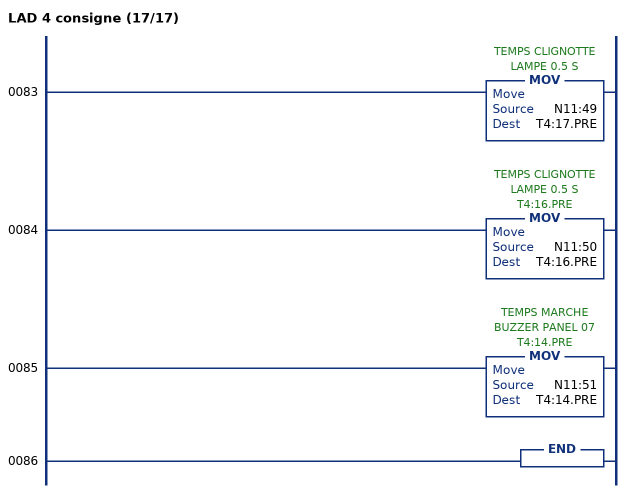
% Rung: 83 %
SOR MOV N11:49 T4:17.PRE EOR
%   N11:49  "TEMPS CLIGNOTTE LAMPE 0.5 S" %
%   T4:17.PRE  "TEMPS CLIGNOTTE LAMPE 0.5 S" %
% Rung: 84 %
SOR MOV N11:50 T4:16.PRE EOR
%   N11:50  "TEMPS CLIGNOTTE LAMPE 0.5 S" %
%   T4:16.PRE  "TEMPS CLIGNOTTE LAMPE 0.5 S T4:16.PRE" %
% Rung: 85 %
SOR MOV N11:51 T4:14.PRE EOR
%   N11:51  "TEMPS MARCHE BUZZER PANEL 07" %
%   T4:14.PRE  "TEMPS MARCHE BUZZER PANEL 07 T4:14.PRE" %
% Rung: 86 %
SOR END EOR

LADDER 5 "communicat"
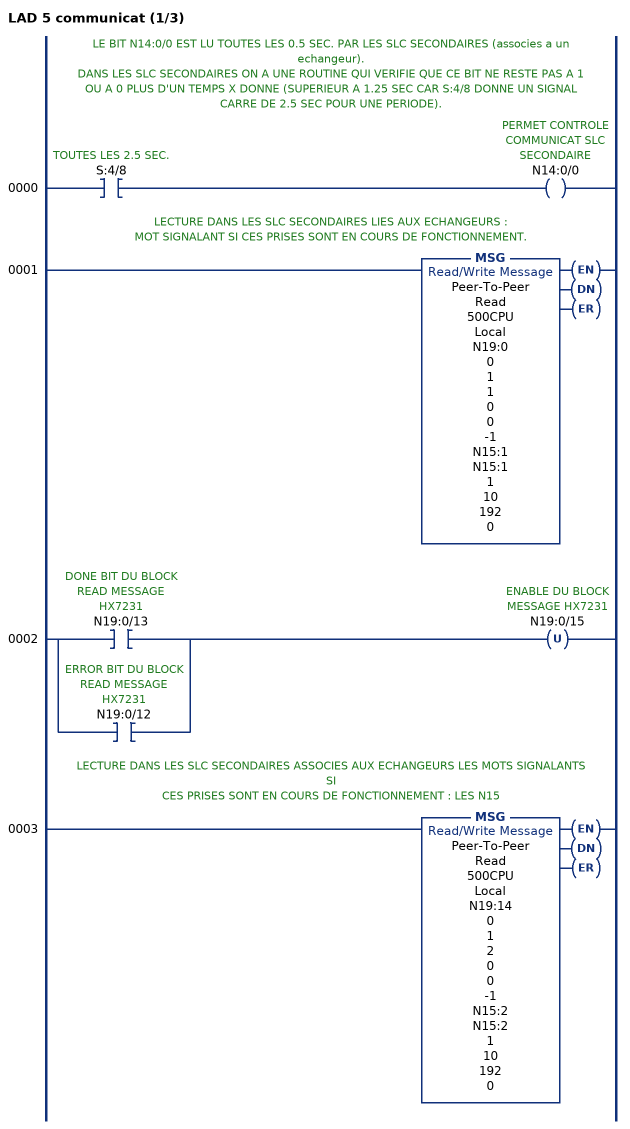
% Rung: 0 %
% LE BIT N14:0/0 EST LU TOUTES LES 0.5 SEC. PAR LES SLC SECONDAIRES (associes a un echangeur).
% DANS LES SLC SECONDAIRES ON A UNE ROUTINE QUI VERIFIE QUE CE BIT NE RESTE PAS A 1 OU A 0 PLUS D'UN TEMPS X DONNE (SUPERIEUR A 1.25 SEC CAR S:4/8 DONNE UN SIGNAL CARRE DE 2.5 SEC POUR UNE PERIODE). %
SOR XIC S:4/8 OTE N14:0/0 EOR
%   S:4/8  "TOUTES LES 2.5 SEC." %
%   N14:0/0  "PERMET CONTROLE COMMUNICAT SLC SECONDAIRE" %
% Rung: 1 %
% LECTURE DANS LES SLC SECONDAIRES LIES AUX ECHANGEURS :
% MOT SIGNALANT SI CES PRISES SONT EN COURS DE FONCTIONNEMENT. %
SOR MSG Peer-To-Peer Read 500CPU Local N19:0 0 1 1 0 0 -1 N15:1 N15:1 1 10 192 0 EOR
%   MSG set-up: 500CPU Read | 10 | 1 | N15:1 | N15:1 | 0 | 1 | 1 | CLIENT | 0 | 0 %
%   N19:0  "LECTURE DU MOT N15:1 DANS HX7231" %
% Rung: 2 %
SOR BST XIC N19:0/13 NXB XIC N19:0/12 BND OTU N19:0/15 EOR
%   N19:0/13  "DONE BIT DU BLOCK READ MESSAGE HX7231" %
%   N19:0/12  "ERROR BIT DU BLOCK READ MESSAGE HX7231" %
%   N19:0/15  "ENABLE DU BLOCK MESSAGE HX7231" %
% Rung: 3 %
% LECTURE DANS LES SLC SECONDAIRES ASSOCIES AUX ECHANGEURS LES MOTS SIGNALANTS SI
% CES PRISES SONT EN COURS DE FONCTIONNEMENT : LES N15 %
SOR MSG Peer-To-Peer Read 500CPU Local N19:14 0 1 2 0 0 -1 N15:2 N15:2 1 10 192 0 EOR
%   MSG set-up: 500CPU Read | 10 | 1 | N15:2 | N15:2 | 0 | 2 | 2 | CLIENT | 0 | 0 %
%   N19:14  "LECTURE DU MOT N15:2 DANS HX7232" %

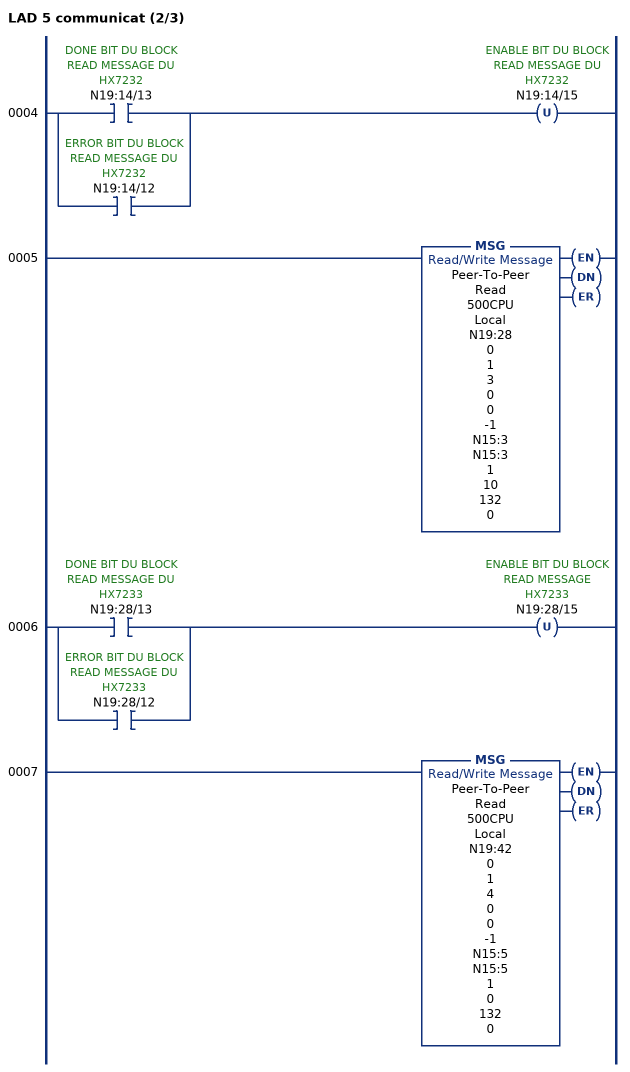
% Rung: 4 %
SOR BST XIC N19:14/13 NXB XIC N19:14/12 BND OTU N19:14/15 EOR
%   N19:14/13  "DONE BIT DU BLOCK READ MESSAGE DU HX7232" %
%   N19:14/12  "ERROR BIT DU BLOCK READ MESSAGE DU HX7232" %
%   N19:14/15  "ENABLE BIT DU BLOCK READ MESSAGE DU HX7232" %
% Rung: 5 %
SOR MSG Peer-To-Peer Read 500CPU Local N19:28 0 1 3 0 0 -1 N15:3 N15:3 1 10 132 0 EOR
%   MSG set-up: 500CPU Read | 10 | 1 | N15:3 | N15:3 | 0 | 3 | 3 | CLIENT | 0 | 0 %
%   N19:28  "LECTURE DU MOT N15:3 (N15:3/1, 2 ET 3) DANS HE7233" %
% Rung: 6 %
SOR BST XIC N19:28/13 NXB XIC N19:28/12 BND OTU N19:28/15 EOR
%   N19:28/13  "DONE BIT DU BLOCK READ MESSAGE DU HX7233" %
%   N19:28/12  "ERROR BIT DU BLOCK READ MESSAGE DU HX7233" %
%   N19:28/15  "ENABLE BIT DU BLOCK READ MESSAGE HX7233" %
% Rung: 7 %
SOR MSG Peer-To-Peer Read 500CPU Local N19:42 0 1 4 0 0 -1 N15:5 N15:5 1 0 132 0 EOR
%   MSG set-up: 500CPU Read | 0 | 1 | N15:5 | N15:5 | 0 | 4 | 4 | CLIENT | 0 | 0 %
%   N19:42  "LECTURE DU MOT N15:5 DANS HX7235" %

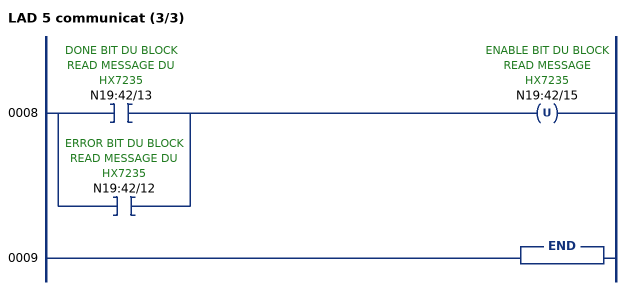
% Rung: 8 %
SOR BST XIC N19:42/13 NXB XIC N19:42/12 BND OTU N19:42/15 EOR
%   N19:42/13  "DONE BIT DU BLOCK READ MESSAGE DU HX7235" %
%   N19:42/12  "ERROR BIT DU BLOCK READ MESSAGE DU HX7235" %
%   N19:42/15  "ENABLE BIT DU BLOCK READ MESSAGE HX7235" %
% Rung: 9 %
SOR END EOR

LADDER 6 "alarmes"
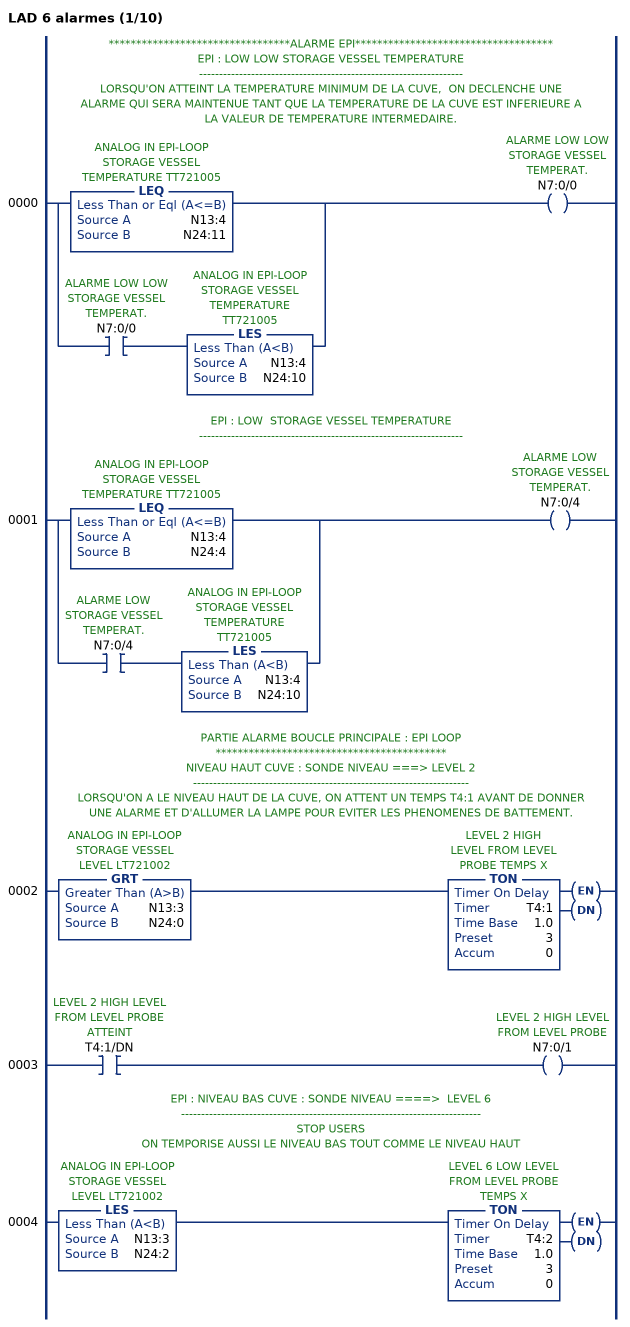
% Rung: 0 %
% *********************************ALARME EPI************************************
% EPI : LOW LOW STORAGE VESSEL TEMPERATURE
% ------------------------------------------------------------------
% LORSQU'ON ATTEINT LA TEMPERATURE MINIMUM DE LA CUVE,  ON DECLENCHE UNE
% ALARME QUI SERA MAINTENUE TANT QUE LA TEMPERATURE DE LA CUVE EST INFERIEURE A
% LA VALEUR DE TEMPERATURE INTERMEDAIRE. %
SOR BST LEQ N13:4 N24:11 NXB XIC N7:0/0 LES N13:4 N24:10 BND OTE N7:0/0 EOR
%   N13:4  "ANALOG IN EPI-LOOP STORAGE VESSEL TEMPERATURE TT721005" %
%   N24:11  "CONSIGNE STORAGE VESSEL LOW LOW TEMPERAT." %
%   N7:0/0  "ALARME LOW LOW STORAGE VESSEL TEMPERAT." %
%   N24:10  "CONSIGNE STORAGE VESSEL INTERMED. TEMPERAT." %
% Rung: 1 %
% EPI : LOW  STORAGE VESSEL TEMPERATURE
% ------------------------------------------------------------------ %
SOR BST LEQ N13:4 N24:4 NXB XIC N7:0/4 LES N13:4 N24:10 BND OTE N7:0/4 EOR
%   N13:4  "ANALOG IN EPI-LOOP STORAGE VESSEL TEMPERATURE TT721005" %
%   N24:4  "CONSIGNE STORAGE VESSEL LOW TEMPERAT." %
%   N7:0/4  "ALARME LOW STORAGE VESSEL TEMPERAT." %
%   N24:10  "CONSIGNE STORAGE VESSEL INTERMED. TEMPERAT." %
% Rung: 2 %
% PARTIE ALARME BOUCLE PRINCIPALE : EPI LOOP
% ******************************************
% NIVEAU HAUT CUVE : SONDE NIVEAU ===> LEVEL 2
% ---------------------------------------------------------------------
% LORSQU'ON A LE NIVEAU HAUT DE LA CUVE, ON ATTENT UN TEMPS T4:1 AVANT DE DONNER
% UNE ALARME ET D'ALLUMER LA LAMPE POUR EVITER LES PHENOMENES DE BATTEMENT. %
SOR GRT N13:3 N24:0 TON T4:1 1.0 3 0 EOR
%   N13:3  "ANALOG IN EPI-LOOP STORAGE VESSEL LEVEL LT721002" %
%   N24:0  "LEVEL 2 HIGH LEVEL FROM LEVEL PROBE" %
%   T4:1  "LEVEL 2 HIGH LEVEL FROM LEVEL PROBE TEMPS X" %
% Rung: 3 %
SOR XIC T4:1/DN OTE N7:0/1 EOR
%   T4:1/DN  "LEVEL 2 HIGH LEVEL FROM LEVEL PROBE ATTEINT" %
%   N7:0/1  "LEVEL 2 HIGH LEVEL FROM LEVEL PROBE" %
% Rung: 4 %
% EPI : NIVEAU BAS CUVE : SONDE NIVEAU ====>  LEVEL 6
% ---------------------------------------------------------------------------
% 
% STOP USERS
% 
% ON TEMPORISE AUSSI LE NIVEAU BAS TOUT COMME LE NIVEAU HAUT %
SOR LES N13:3 N24:2 TON T4:2 1.0 3 0 EOR
%   N13:3  "ANALOG IN EPI-LOOP STORAGE VESSEL LEVEL LT721002" %
%   N24:2  "LEVEL 6 LOW LEVEL FROM LEVEL PROBE" %
%   T4:2  "LEVEL 6 LOW LEVEL FROM LEVEL PROBE TEMPS X" %

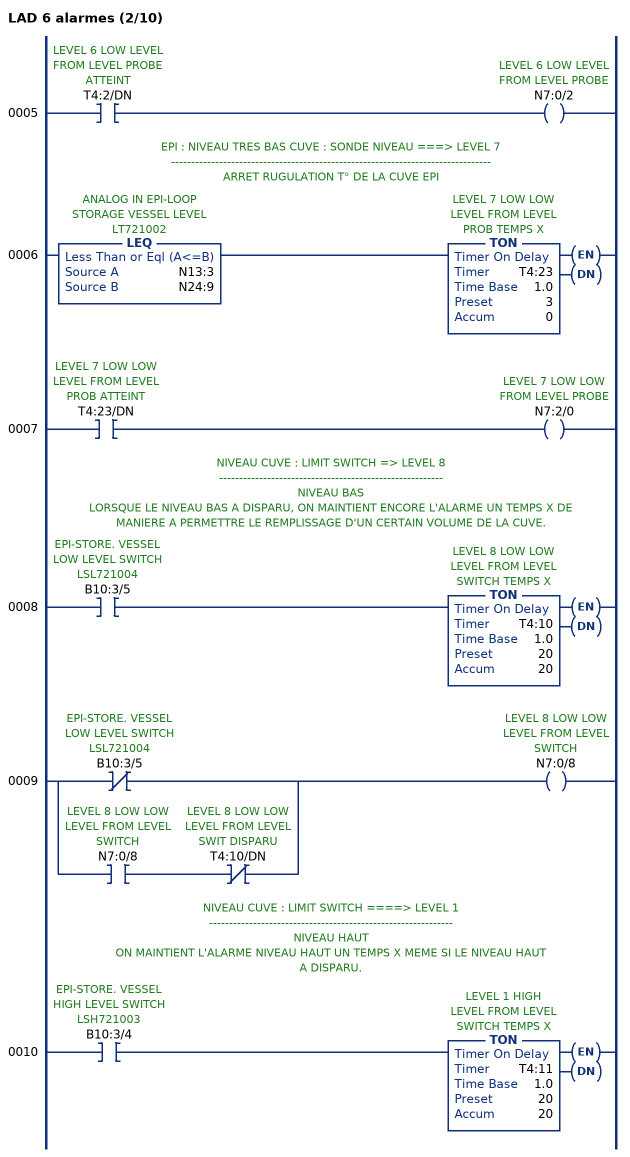
% Rung: 5 %
SOR XIC T4:2/DN OTE N7:0/2 EOR
%   T4:2/DN  "LEVEL 6 LOW LEVEL FROM LEVEL PROBE ATTEINT" %
%   N7:0/2  "LEVEL 6 LOW LEVEL FROM LEVEL PROBE" %
% Rung: 6 %
% EPI : NIVEAU TRES BAS CUVE : SONDE NIVEAU ===> LEVEL 7
% --------------------------------------------------------------------------------
% 
% ARRET RUGULATION T° DE LA CUVE EPI %
SOR LEQ N13:3 N24:9 TON T4:23 1.0 3 0 EOR
%   N13:3  "ANALOG IN EPI-LOOP STORAGE VESSEL LEVEL LT721002" %
%   N24:9  "LEVEL 7 LOW LOW LEVEL FROM LEVEL PROBE" %
%   T4:23  "LEVEL 7 LOW LOW LEVEL FROM LEVEL PROB TEMPS X" %
% Rung: 7 %
SOR XIC T4:23/DN OTE N7:2/0 EOR
%   T4:23/DN  "LEVEL 7 LOW LOW LEVEL FROM LEVEL PROB ATTEINT" %
%   N7:2/0  "LEVEL 7 LOW LOW FROM LEVEL PROBE" %
% Rung: 8 %
% NIVEAU CUVE : LIMIT SWITCH => LEVEL 8
% --------------------------------------------------------
% NIVEAU BAS
% 
% LORSQUE LE NIVEAU BAS A DISPARU, ON MAINTIENT ENCORE L'ALARME UN TEMPS X DE
% MANIERE A PERMETTRE LE REMPLISSAGE D'UN CERTAIN VOLUME DE LA CUVE. %
SOR XIC B10:3/5 TON T4:10 1.0 20 20 EOR
%   B10:3/5  "EPI-STORE. VESSEL LOW LEVEL SWITCH LSL721004" %
%   T4:10  "LEVEL 8 LOW LOW LEVEL FROM LEVEL SWITCH TEMPS X" %
% Rung: 9 %
SOR BST XIO B10:3/5 NXB XIC N7:0/8 XIO T4:10/DN BND OTE N7:0/8 EOR
%   B10:3/5  "EPI-STORE. VESSEL LOW LEVEL SWITCH LSL721004" %
%   N7:0/8  "LEVEL 8 LOW LOW LEVEL FROM LEVEL SWITCH" %
%   T4:10/DN  "LEVEL 8 LOW LOW LEVEL FROM LEVEL SWIT DISPARU" %
% Rung: 10 %
% NIVEAU CUVE : LIMIT SWITCH ====> LEVEL 1
% -------------------------------------------------------------
% NIVEAU HAUT
% 
% ON MAINTIENT L'ALARME NIVEAU HAUT UN TEMPS X MEME SI LE NIVEAU HAUT
% A DISPARU. %
SOR XIC B10:3/4 TON T4:11 1.0 20 20 EOR
%   B10:3/4  "EPI-STORE. VESSEL HIGH LEVEL SWITCH LSH721003" %
%   T4:11  "LEVEL 1 HIGH LEVEL FROM LEVEL SWITCH TEMPS X" %

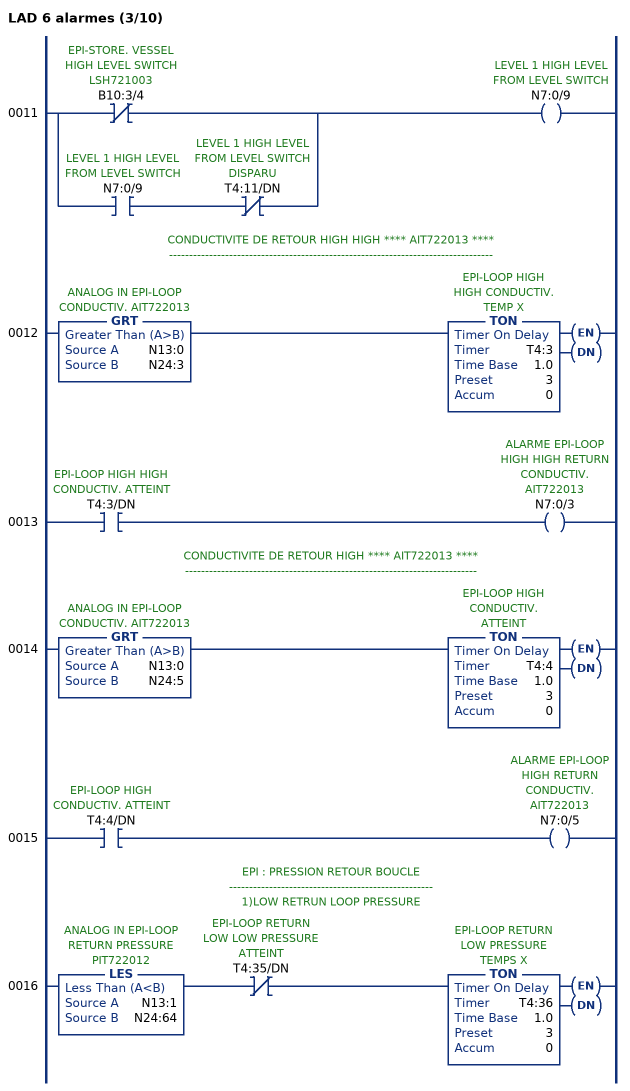
% Rung: 11 %
SOR BST XIO B10:3/4 NXB XIC N7:0/9 XIO T4:11/DN BND OTE N7:0/9 EOR
%   B10:3/4  "EPI-STORE. VESSEL HIGH LEVEL SWITCH LSH721003" %
%   N7:0/9  "LEVEL 1 HIGH LEVEL FROM LEVEL SWITCH" %
%   T4:11/DN  "LEVEL 1 HIGH LEVEL FROM LEVEL SWITCH DISPARU" %
% Rung: 12 %
% CONDUCTIVITE DE RETOUR HIGH HIGH **** AIT722013 ****
% --------------------------------------------------------------------------------- %
SOR GRT N13:0 N24:3 TON T4:3 1.0 3 0 EOR
%   N13:0  "ANALOG IN EPI-LOOP CONDUCTIV. AIT722013" %
%   N24:3  "CONSIGNE HIGH HIGH RETURN CONDUCT. AIT722013" %
%   T4:3  "EPI-LOOP HIGH HIGH CONDUCTIV. TEMP X" %
% Rung: 13 %
SOR XIC T4:3/DN OTE N7:0/3 EOR
%   T4:3/DN  "EPI-LOOP HIGH HIGH CONDUCTIV. ATTEINT" %
%   N7:0/3  "ALARME EPI-LOOP HIGH HIGH RETURN CONDUCTIV. AIT722013" %
% Rung: 14 %
% CONDUCTIVITE DE RETOUR HIGH **** AIT722013 ****
% ------------------------------------------------------------------------- %
SOR GRT N13:0 N24:5 TON T4:4 1.0 3 0 EOR
%   N13:0  "ANALOG IN EPI-LOOP CONDUCTIV. AIT722013" %
%   N24:5  "CONSIGNE HIGH RETURN CONDUCT. AIT722013" %
%   T4:4  "EPI-LOOP HIGH CONDUCTIV. ATTEINT" %
% Rung: 15 %
SOR XIC T4:4/DN OTE N7:0/5 EOR
%   T4:4/DN  "EPI-LOOP HIGH CONDUCTIV. ATTEINT" %
%   N7:0/5  "ALARME EPI-LOOP HIGH RETURN CONDUCTIV. AIT722013" %
% Rung: 16 %
% EPI : PRESSION RETOUR BOUCLE
% ---------------------------------------------------
% 1)LOW RETRUN LOOP PRESSURE %
SOR LES N13:1 N24:64 XIO T4:35/DN TON T4:36 1.0 3 0 EOR
%   N13:1  "ANALOG IN EPI-LOOP RETURN PRESSURE PIT722012" %
%   N24:64  "PRESSION LOW RETOUR BOUCLE" %
%   T4:35/DN  "EPI-LOOP RETURN LOW LOW PRESSURE ATTEINT" %
%   T4:36  "EPI-LOOP RETURN LOW PRESSURE TEMPS X" %

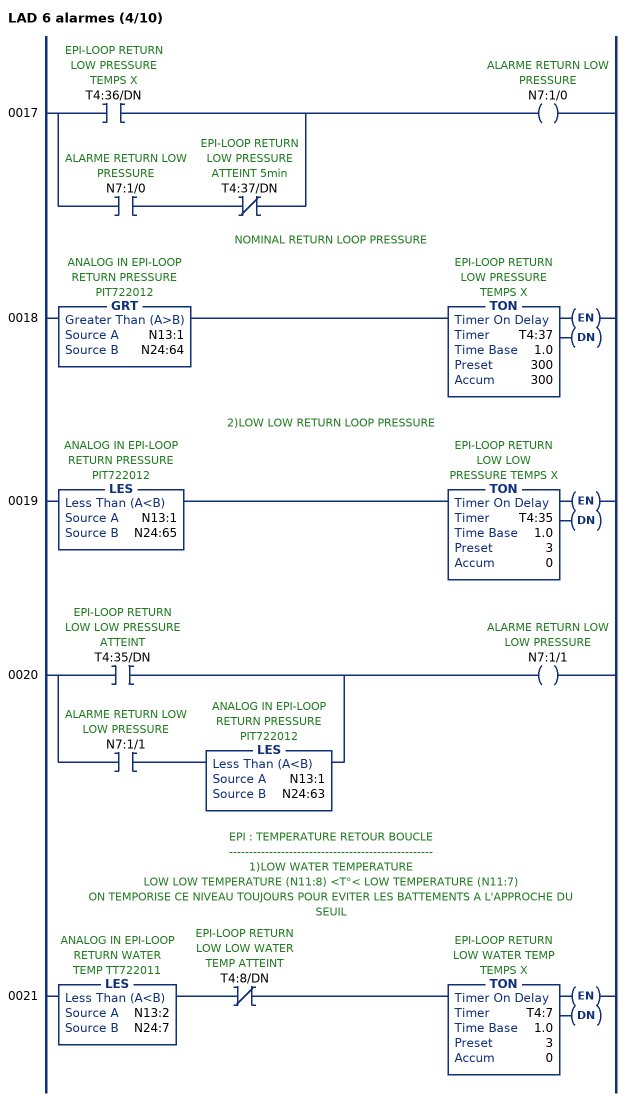
% Rung: 17 %
SOR BST XIC T4:36/DN NXB XIC N7:1/0 XIO T4:37/DN BND OTE N7:1/0 EOR
%   T4:36/DN  "EPI-LOOP RETURN LOW PRESSURE TEMPS X" %
%   N7:1/0  "ALARME RETURN LOW PRESSURE" %
%   T4:37/DN  "EPI-LOOP RETURN LOW PRESSURE ATTEINT 5min" %
% Rung: 18 %
% NOMINAL RETURN LOOP PRESSURE %
SOR GRT N13:1 N24:64 TON T4:37 1.0 300 300 EOR
%   N13:1  "ANALOG IN EPI-LOOP RETURN PRESSURE PIT722012" %
%   N24:64  "PRESSION LOW RETOUR BOUCLE" %
%   T4:37  "EPI-LOOP RETURN LOW PRESSURE TEMPS X" %
% Rung: 19 %
% 2)LOW LOW RETURN LOOP PRESSURE %
SOR LES N13:1 N24:65 TON T4:35 1.0 3 0 EOR
%   N13:1  "ANALOG IN EPI-LOOP RETURN PRESSURE PIT722012" %
%   N24:65  "PRESSION LOW LOW RETOUR BOUCLE" %
%   T4:35  "EPI-LOOP RETURN LOW LOW PRESSURE TEMPS X" %
% Rung: 20 %
SOR BST XIC T4:35/DN NXB XIC N7:1/1 LES N13:1 N24:63 BND OTE N7:1/1 EOR
%   T4:35/DN  "EPI-LOOP RETURN LOW LOW PRESSURE ATTEINT" %
%   N7:1/1  "ALARME RETURN LOW LOW PRESSURE" %
%   N13:1  "ANALOG IN EPI-LOOP RETURN PRESSURE PIT722012" %
%   N24:63  "PRESSION NOMINALE RETOUR BOUCLE" %
% Rung: 21 %
% EPI : TEMPERATURE RETOUR BOUCLE
% ---------------------------------------------------
% 1)LOW WATER TEMPERATURE
% 
% LOW LOW TEMPERATURE (N11:8) <T°< LOW TEMPERATURE (N11:7)
% ON TEMPORISE CE NIVEAU TOUJOURS POUR EVITER LES BATTEMENTS A L'APPROCHE DU SEUIL %
SOR LES N13:2 N24:7 XIO T4:8/DN TON T4:7 1.0 3 0 EOR
%   N13:2  "ANALOG IN EPI-LOOP RETURN WATER TEMP TT722011" %
%   N24:7  "CONSIGNE LOW LOOP RETURN TEMPERAT." %
%   T4:8/DN  "EPI-LOOP RETURN LOW LOW WATER TEMP ATTEINT" %
%   T4:7  "EPI-LOOP RETURN LOW WATER TEMP TEMPS X" %

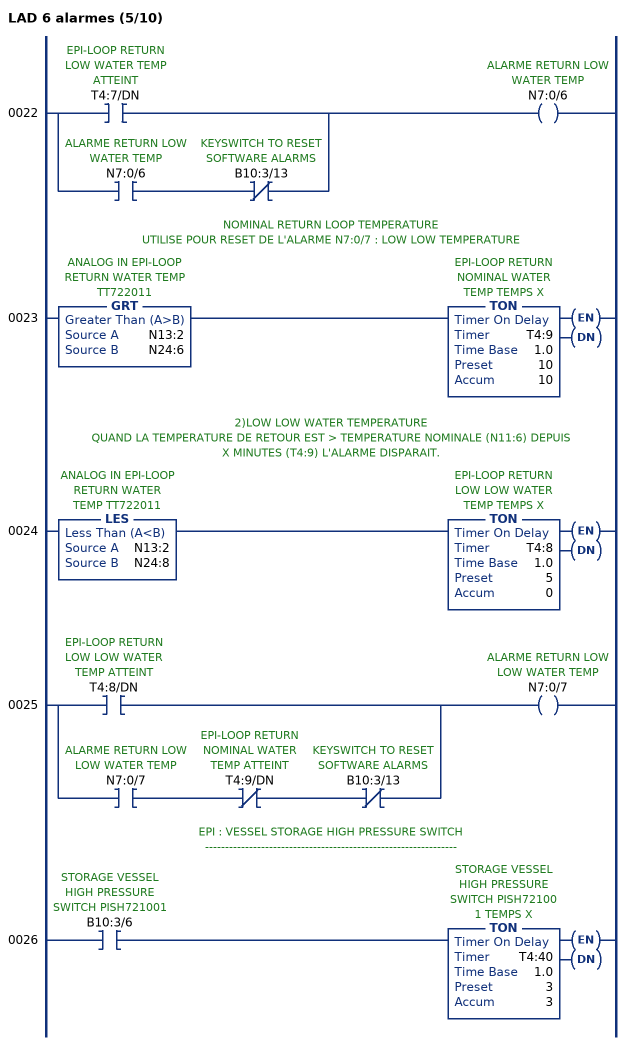
% Rung: 22 %
SOR BST XIC T4:7/DN NXB XIC N7:0/6 XIO B10:3/13 BND OTE N7:0/6 EOR
%   T4:7/DN  "EPI-LOOP RETURN LOW WATER TEMP ATTEINT" %
%   N7:0/6  "ALARME RETURN LOW WATER TEMP" %
%   B10:3/13  "KEYSWITCH TO RESET SOFTWARE ALARMS" %
% Rung: 23 %
% NOMINAL RETURN LOOP TEMPERATURE
% 
% UTILISE POUR RESET DE L'ALARME N7:0/7 : LOW LOW TEMPERATURE %
SOR GRT N13:2 N24:6 TON T4:9 1.0 10 10 EOR
%   N13:2  "ANALOG IN EPI-LOOP RETURN WATER TEMP TT722011" %
%   N24:6  "CONSIGNE NOMINAL RETURN TEMPERAT." %
%   T4:9  "EPI-LOOP RETURN NOMINAL WATER TEMP TEMPS X" %
% Rung: 24 %
% 2)LOW LOW WATER TEMPERATURE
% 
% QUAND LA TEMPERATURE DE RETOUR EST > TEMPERATURE NOMINALE (N11:6) DEPUIS
% X MINUTES (T4:9) L'ALARME DISPARAIT. %
SOR LES N13:2 N24:8 TON T4:8 1.0 5 0 EOR
%   N13:2  "ANALOG IN EPI-LOOP RETURN WATER TEMP TT722011" %
%   N24:8  "CONSIGNE LOW LOW LOOP RETURN TEMPERAT." %
%   T4:8  "EPI-LOOP RETURN LOW LOW WATER TEMP TEMPS X" %
% Rung: 25 %
SOR BST XIC T4:8/DN NXB XIC N7:0/7 XIO T4:9/DN XIO B10:3/13 BND OTE N7:0/7 EOR
%   T4:8/DN  "EPI-LOOP RETURN LOW LOW WATER TEMP ATTEINT" %
%   N7:0/7  "ALARME RETURN LOW LOW WATER TEMP" %
%   T4:9/DN  "EPI-LOOP RETURN NOMINAL WATER TEMP ATTEINT" %
%   B10:3/13  "KEYSWITCH TO RESET SOFTWARE ALARMS" %
% Rung: 26 %
% EPI : VESSEL STORAGE HIGH PRESSURE SWITCH
% --------------------------------------------------------------- %
SOR XIC B10:3/6 TON T4:40 1.0 3 3 EOR
%   B10:3/6  "STORAGE VESSEL HIGH PRESSURE SWITCH PISH721001" %
%   T4:40  "STORAGE VESSEL HIGH PRESSURE SWITCH PISH721001 TEMPS X" %

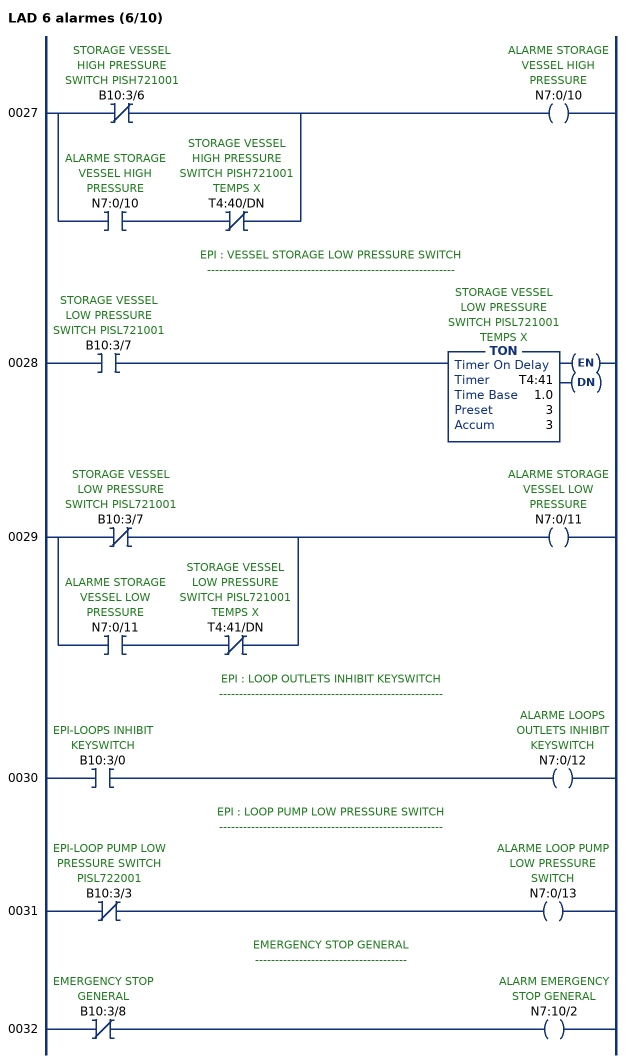
% Rung: 27 %
SOR BST XIO B10:3/6 NXB XIC N7:0/10 XIO T4:40/DN BND OTE N7:0/10 EOR
%   B10:3/6  "STORAGE VESSEL HIGH PRESSURE SWITCH PISH721001" %
%   N7:0/10  "ALARME STORAGE VESSEL HIGH PRESSURE" %
%   T4:40/DN  "STORAGE VESSEL HIGH PRESSURE SWITCH PISH721001 TEMPS X" %
% Rung: 28 %
% EPI : VESSEL STORAGE LOW PRESSURE SWITCH
% -------------------------------------------------------------- %
SOR XIC B10:3/7 TON T4:41 1.0 3 3 EOR
%   B10:3/7  "STORAGE VESSEL LOW PRESSURE SWITCH PISL721001" %
%   T4:41  "STORAGE VESSEL LOW PRESSURE SWITCH PISL721001 TEMPS X" %
% Rung: 29 %
SOR BST XIO B10:3/7 NXB XIC N7:0/11 XIO T4:41/DN BND OTE N7:0/11 EOR
%   B10:3/7  "STORAGE VESSEL LOW PRESSURE SWITCH PISL721001" %
%   N7:0/11  "ALARME STORAGE VESSEL LOW PRESSURE" %
%   T4:41/DN  "STORAGE VESSEL LOW PRESSURE SWITCH PISL721001 TEMPS X" %
% Rung: 30 %
% EPI : LOOP OUTLETS INHIBIT KEYSWITCH
% -------------------------------------------------------- %
SOR XIC B10:3/0 OTE N7:0/12 EOR
%   B10:3/0  "EPI-LOOPS INHIBIT KEYSWITCH" %
%   N7:0/12  "ALARME LOOPS OUTLETS INHIBIT KEYSWITCH" %
% Rung: 31 %
% EPI : LOOP PUMP LOW PRESSURE SWITCH
% -------------------------------------------------------- %
SOR XIO B10:3/3 OTE N7:0/13 EOR
%   B10:3/3  "EPI-LOOP PUMP LOW PRESSURE SWITCH PISL722001" %
%   N7:0/13  "ALARME LOOP PUMP LOW PRESSURE SWITCH" %
% Rung: 32 %
% EMERGENCY STOP GENERAL
% -------------------------------------- %
SOR XIO B10:3/8 OTE N7:10/2 EOR
%   B10:3/8  "EMERGENCY STOP GENERAL" %
%   N7:10/2  "ALARM EMERGENCY STOP GENERAL" %

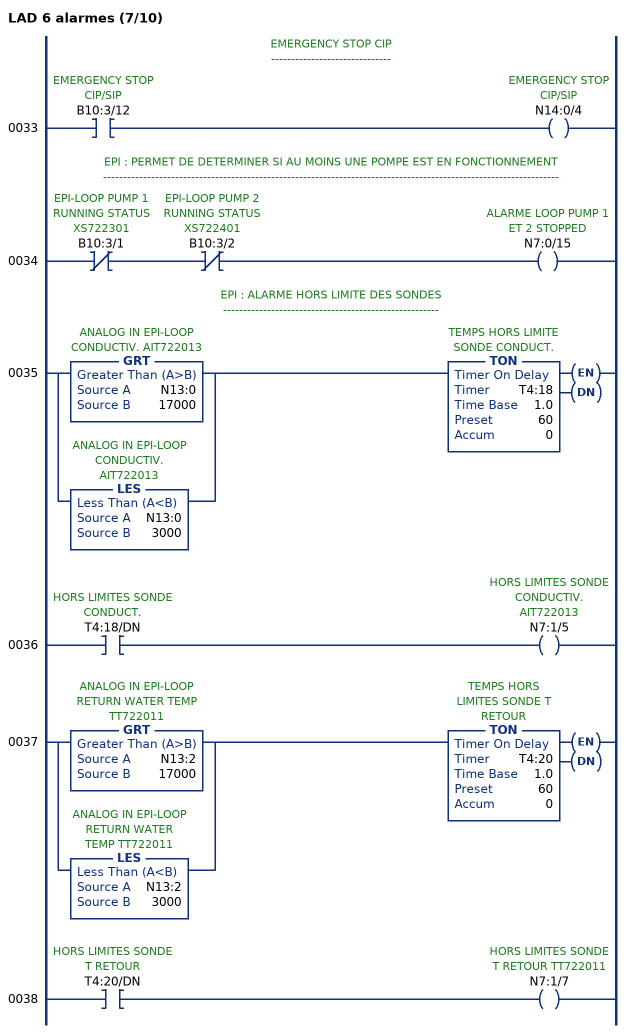
% Rung: 33 %
% EMERGENCY STOP CIP
% ------------------------------ %
SOR XIC B10:3/12 OTE N14:0/4 EOR
%   B10:3/12  "EMERGENCY STOP CIP/SIP" %
%   N14:0/4  "EMERGENCY STOP CIP/SIP" %
% Rung: 34 %
% EPI : PERMET DE DETERMINER SI AU MOINS UNE POMPE EST EN FONCTIONNEMENT
% ------------------------------------------------------------------------------------------------------------------ %
SOR XIO B10:3/1 XIO B10:3/2 OTE N7:0/15 EOR
%   B10:3/1  "EPI-LOOP PUMP 1 RUNNING STATUS XS722301" %
%   B10:3/2  "EPI-LOOP PUMP 2 RUNNING STATUS XS722401" %
%   N7:0/15  "ALARME LOOP PUMP 1 ET 2 STOPPED" %
% Rung: 35 %
% EPI : ALARME HORS LIMITE DES SONDES
% ------------------------------------------------------ %
SOR BST GRT N13:0 17000 NXB LES N13:0 3000 BND TON T4:18 1.0 60 0 EOR
%   N13:0  "ANALOG IN EPI-LOOP CONDUCTIV. AIT722013" %
%   T4:18  "TEMPS HORS LIMITE SONDE CONDUCT." %
% Rung: 36 %
SOR XIC T4:18/DN OTE N7:1/5 EOR
%   T4:18/DN  "HORS LIMITES SONDE CONDUCT." %
%   N7:1/5  "HORS LIMITES SONDE CONDUCTIV. AIT722013" %
% Rung: 37 %
SOR BST GRT N13:2 17000 NXB LES N13:2 3000 BND TON T4:20 1.0 60 0 EOR
%   N13:2  "ANALOG IN EPI-LOOP RETURN WATER TEMP TT722011" %
%   T4:20  "TEMPS HORS LIMITES SONDE T RETOUR" %
% Rung: 38 %
SOR XIC T4:20/DN OTE N7:1/7 EOR
%   T4:20/DN  "HORS LIMITES SONDE T RETOUR" %
%   N7:1/7  "HORS LIMITES SONDE T RETOUR TT722011" %

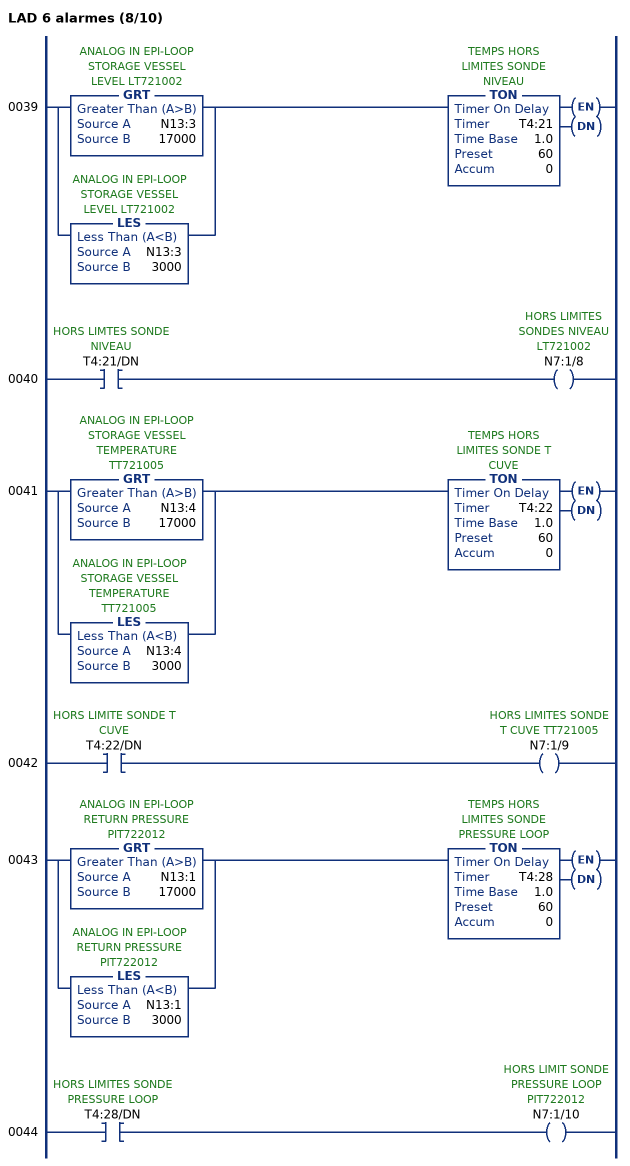
% Rung: 39 %
SOR BST GRT N13:3 17000 NXB LES N13:3 3000 BND TON T4:21 1.0 60 0 EOR
%   N13:3  "ANALOG IN EPI-LOOP STORAGE VESSEL LEVEL LT721002" %
%   T4:21  "TEMPS HORS LIMITES SONDE NIVEAU" %
% Rung: 40 %
SOR XIC T4:21/DN OTE N7:1/8 EOR
%   T4:21/DN  "HORS LIMTES SONDE NIVEAU" %
%   N7:1/8  "HORS LIMITES SONDES NIVEAU LT721002" %
% Rung: 41 %
SOR BST GRT N13:4 17000 NXB LES N13:4 3000 BND TON T4:22 1.0 60 0 EOR
%   N13:4  "ANALOG IN EPI-LOOP STORAGE VESSEL TEMPERATURE TT721005" %
%   T4:22  "TEMPS HORS LIMITES SONDE T CUVE" %
% Rung: 42 %
SOR XIC T4:22/DN OTE N7:1/9 EOR
%   T4:22/DN  "HORS LIMITE SONDE T CUVE" %
%   N7:1/9  "HORS LIMITES SONDE T CUVE TT721005" %
% Rung: 43 %
SOR BST GRT N13:1 17000 NXB LES N13:1 3000 BND TON T4:28 1.0 60 0 EOR
%   N13:1  "ANALOG IN EPI-LOOP RETURN PRESSURE PIT722012" %
%   T4:28  "TEMPS HORS LIMITES SONDE PRESSURE LOOP" %
% Rung: 44 %
SOR XIC T4:28/DN OTE N7:1/10 EOR
%   T4:28/DN  "HORS LIMITES SONDE PRESSURE LOOP" %
%   N7:1/10  "HORS LIMIT SONDE PRESSURE LOOP PIT722012" %

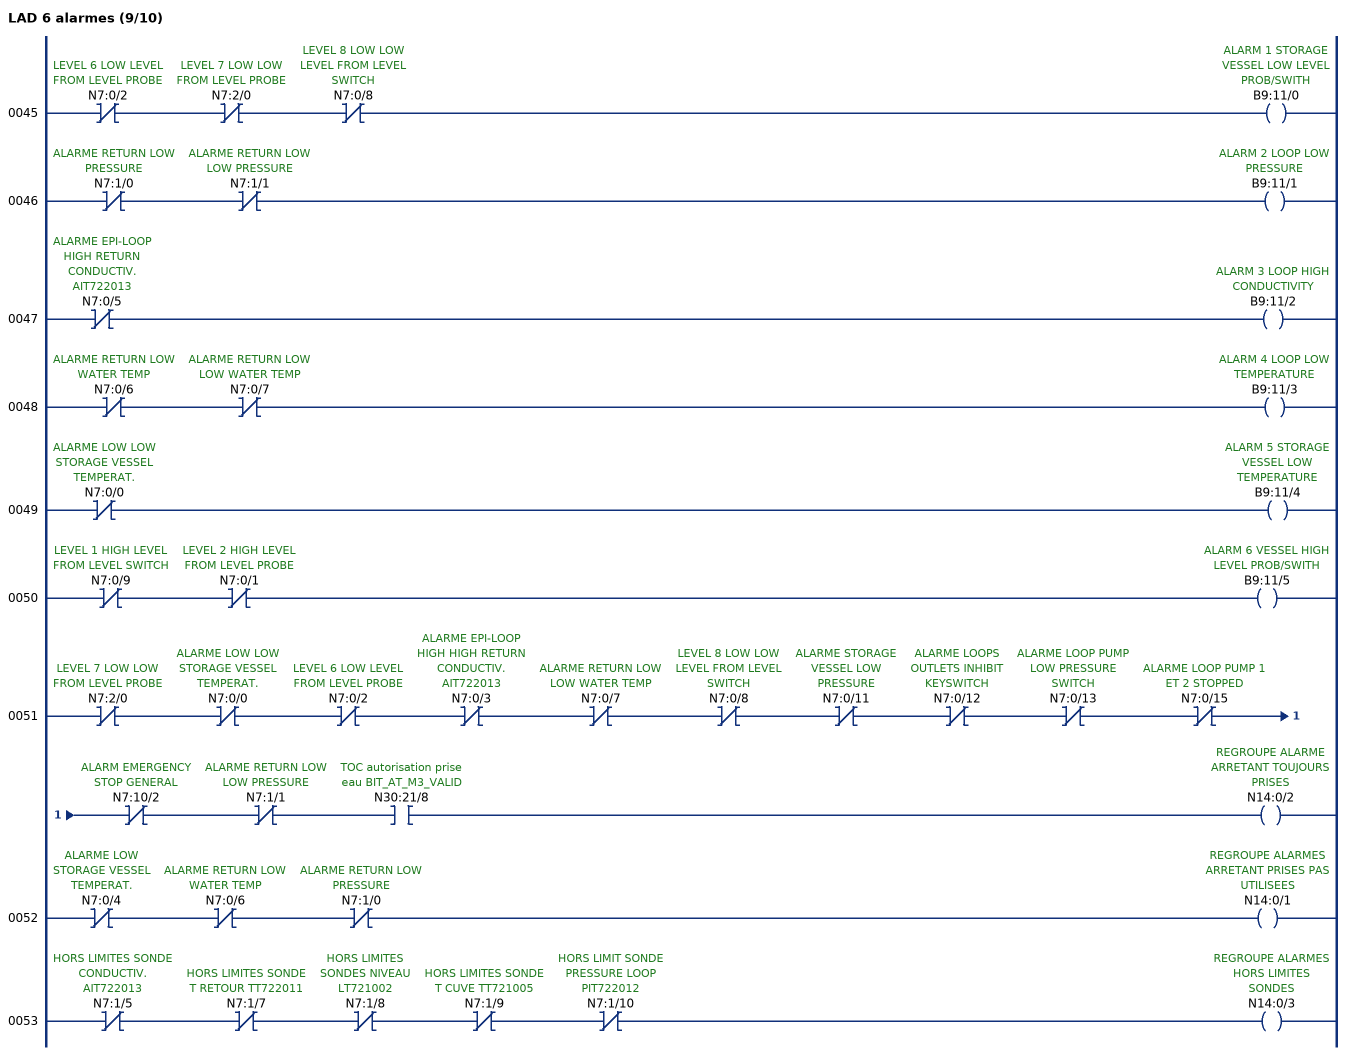
% Rung: 45 %
SOR XIO N7:0/2 XIO N7:2/0 XIO N7:0/8 OTE B9:11/0 EOR
%   N7:0/2  "LEVEL 6 LOW LEVEL FROM LEVEL PROBE" %
%   N7:2/0  "LEVEL 7 LOW LOW FROM LEVEL PROBE" %
%   N7:0/8  "LEVEL 8 LOW LOW LEVEL FROM LEVEL SWITCH" %
%   B9:11/0  "ALARM 1 STORAGE VESSEL LOW LEVEL PROB/SWITH" %
% Rung: 46 %
SOR XIO N7:1/0 XIO N7:1/1 OTE B9:11/1 EOR
%   N7:1/0  "ALARME RETURN LOW PRESSURE" %
%   N7:1/1  "ALARME RETURN LOW LOW PRESSURE" %
%   B9:11/1  "ALARM 2 LOOP LOW PRESSURE" %
% Rung: 47 %
SOR XIO N7:0/5 OTE B9:11/2 EOR
%   N7:0/5  "ALARME EPI-LOOP HIGH RETURN CONDUCTIV. AIT722013" %
%   B9:11/2  "ALARM 3 LOOP HIGH CONDUCTIVITY" %
% Rung: 48 %
SOR XIO N7:0/6 XIO N7:0/7 OTE B9:11/3 EOR
%   N7:0/6  "ALARME RETURN LOW WATER TEMP" %
%   N7:0/7  "ALARME RETURN LOW LOW WATER TEMP" %
%   B9:11/3  "ALARM 4 LOOP LOW TEMPERATURE" %
% Rung: 49 %
SOR XIO N7:0/0 OTE B9:11/4 EOR
%   N7:0/0  "ALARME LOW LOW STORAGE VESSEL TEMPERAT." %
%   B9:11/4  "ALARM 5 STORAGE VESSEL LOW TEMPERATURE" %
% Rung: 50 %
SOR XIO N7:0/9 XIO N7:0/1 OTE B9:11/5 EOR
%   N7:0/9  "LEVEL 1 HIGH LEVEL FROM LEVEL SWITCH" %
%   N7:0/1  "LEVEL 2 HIGH LEVEL FROM LEVEL PROBE" %
%   B9:11/5  "ALARM 6 VESSEL HIGH LEVEL PROB/SWITH" %
% Rung: 51 %
SOR XIO N7:2/0 XIO N7:0/0 XIO N7:0/2 XIO N7:0/3 XIO N7:0/7 XIO N7:0/8 XIO N7:0/11 XIO N7:0/12 XIO N7:0/13 XIO N7:0/15 XIO N7:10/2 XIO N7:1/1 XIC N30:21/8 OTE N14:0/2 EOR
%   N7:2/0  "LEVEL 7 LOW LOW FROM LEVEL PROBE" %
%   N7:0/0  "ALARME LOW LOW STORAGE VESSEL TEMPERAT." %
%   N7:0/2  "LEVEL 6 LOW LEVEL FROM LEVEL PROBE" %
%   N7:0/3  "ALARME EPI-LOOP HIGH HIGH RETURN CONDUCTIV. AIT722013" %
%   N7:0/7  "ALARME RETURN LOW LOW WATER TEMP" %
%   N7:0/8  "LEVEL 8 LOW LOW LEVEL FROM LEVEL SWITCH" %
%   N7:0/11  "ALARME STORAGE VESSEL LOW PRESSURE" %
%   N7:0/12  "ALARME LOOPS OUTLETS INHIBIT KEYSWITCH" %
%   N7:0/13  "ALARME LOOP PUMP LOW PRESSURE SWITCH" %
%   N7:0/15  "ALARME LOOP PUMP 1 ET 2 STOPPED" %
%   N7:10/2  "ALARM EMERGENCY STOP GENERAL" %
%   N7:1/1  "ALARME RETURN LOW LOW PRESSURE" %
%   N30:21/8  BIT_AT_M3_VALID  "TOC autorisation prise eau" %
%   N14:0/2  "REGROUPE ALARME ARRETANT TOUJOURS PRISES" %
% Rung: 52 %
SOR XIO N7:0/4 XIO N7:0/6 XIO N7:1/0 OTE N14:0/1 EOR
%   N7:0/4  "ALARME LOW STORAGE VESSEL TEMPERAT." %
%   N7:0/6  "ALARME RETURN LOW WATER TEMP" %
%   N7:1/0  "ALARME RETURN LOW PRESSURE" %
%   N14:0/1  "REGROUPE ALARMES ARRETANT PRISES PAS UTILISEES" %
% Rung: 53 %
SOR XIO N7:1/5 XIO N7:1/7 XIO N7:1/8 XIO N7:1/9 XIO N7:1/10 OTE N14:0/3 EOR
%   N7:1/5  "HORS LIMITES SONDE CONDUCTIV. AIT722013" %
%   N7:1/7  "HORS LIMITES SONDE T RETOUR TT722011" %
%   N7:1/8  "HORS LIMITES SONDES NIVEAU LT721002" %
%   N7:1/9  "HORS LIMITES SONDE T CUVE TT721005" %
%   N7:1/10  "HORS LIMIT SONDE PRESSURE LOOP PIT722012" %
%   N14:0/3  "REGROUPE ALARMES HORS LIMITES SONDES" %

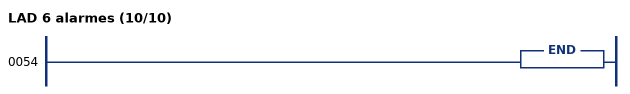
% Rung: 54 %
SOR END EOR

LADDER 7 "programme"
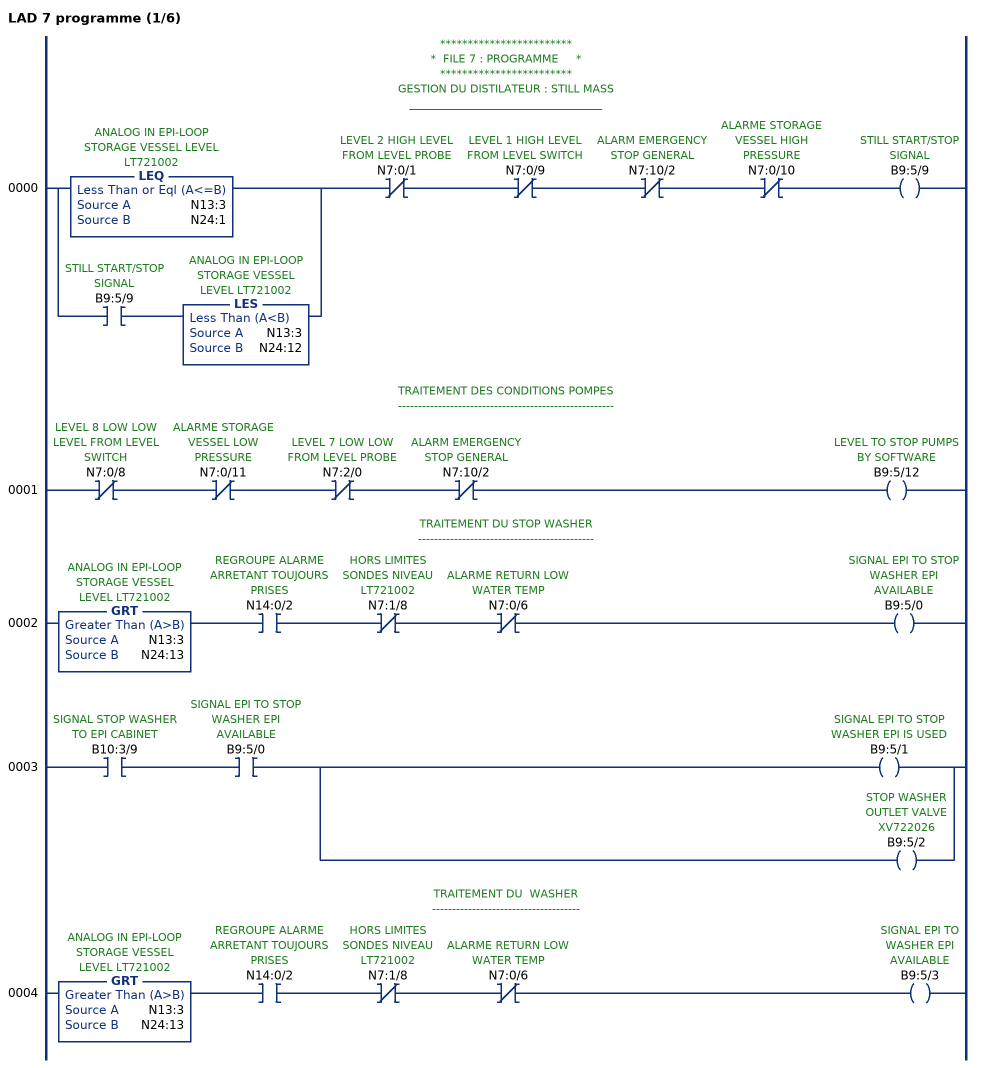
% Rung: 0 %
% ************************
% *  FILE 7 : PROGRAMME     *
% ************************
% GESTION DU DISTILATEUR : STILL MASS
% ___________________________________ %
SOR BST LEQ N13:3 N24:1 NXB XIC B9:5/9 LES N13:3 N24:12 BND XIO N7:0/1 XIO N7:0/9 XIO N7:10/2 XIO N7:0/10 OTE B9:5/9 EOR
%   N13:3  "ANALOG IN EPI-LOOP STORAGE VESSEL LEVEL LT721002" %
%   N24:1  "LEVEL 4 LEVEL FROM LEVEL PROBE START STIL" %
%   B9:5/9  "STILL START/STOP SIGNAL" %
%   N24:12  "LEVEL 3 LEVEL FROM LEVEL PROBE STOP STILL" %
%   N7:0/1  "LEVEL 2 HIGH LEVEL FROM LEVEL PROBE" %
%   N7:0/9  "LEVEL 1 HIGH LEVEL FROM LEVEL SWITCH" %
%   N7:10/2  "ALARM EMERGENCY STOP GENERAL" %
%   N7:0/10  "ALARME STORAGE VESSEL HIGH PRESSURE" %
% Rung: 1 %
% TRAITEMENT DES CONDITIONS POMPES
% ------------------------------------------------------ %
SOR XIO N7:0/8 XIO N7:0/11 XIO N7:2/0 XIO N7:10/2 OTE B9:5/12 EOR
%   N7:0/8  "LEVEL 8 LOW LOW LEVEL FROM LEVEL SWITCH" %
%   N7:0/11  "ALARME STORAGE VESSEL LOW PRESSURE" %
%   N7:2/0  "LEVEL 7 LOW LOW FROM LEVEL PROBE" %
%   N7:10/2  "ALARM EMERGENCY STOP GENERAL" %
%   B9:5/12  "LEVEL TO STOP PUMPS BY SOFTWARE" %
% Rung: 2 %
% TRAITEMENT DU STOP WASHER
% -------------------------------------------- %
SOR GRT N13:3 N24:13 XIC N14:0/2 XIO N7:1/8 XIO N7:0/6 OTE B9:5/0 EOR
%   N13:3  "ANALOG IN EPI-LOOP STORAGE VESSEL LEVEL LT721002" %
%   N24:13  "LEVEL 5 LEVEL FROM LEVEL PROB AUTHORISE CIP+WASH.M" %
%   N14:0/2  "REGROUPE ALARME ARRETANT TOUJOURS PRISES" %
%   N7:1/8  "HORS LIMITES SONDES NIVEAU LT721002" %
%   N7:0/6  "ALARME RETURN LOW WATER TEMP" %
%   B9:5/0  "SIGNAL EPI TO STOP WASHER EPI AVAILABLE" %
% Rung: 3 %
SOR XIC B10:3/9 XIC B9:5/0 BST OTE B9:5/1 NXB OTE B9:5/2 BND EOR
%   B10:3/9  "SIGNAL STOP WASHER TO EPI CABINET" %
%   B9:5/0  "SIGNAL EPI TO STOP WASHER EPI AVAILABLE" %
%   B9:5/1  "SIGNAL EPI TO STOP WASHER EPI IS USED" %
%   B9:5/2  "STOP WASHER OUTLET VALVE XV722026" %
% Rung: 4 %
% TRAITEMENT DU  WASHER
% ------------------------------------- %
SOR GRT N13:3 N24:13 XIC N14:0/2 XIO N7:1/8 XIO N7:0/6 OTE B9:5/3 EOR
%   N13:3  "ANALOG IN EPI-LOOP STORAGE VESSEL LEVEL LT721002" %
%   N24:13  "LEVEL 5 LEVEL FROM LEVEL PROB AUTHORISE CIP+WASH.M" %
%   N14:0/2  "REGROUPE ALARME ARRETANT TOUJOURS PRISES" %
%   N7:1/8  "HORS LIMITES SONDES NIVEAU LT721002" %
%   N7:0/6  "ALARME RETURN LOW WATER TEMP" %
%   B9:5/3  "SIGNAL EPI TO WASHER EPI AVAILABLE" %

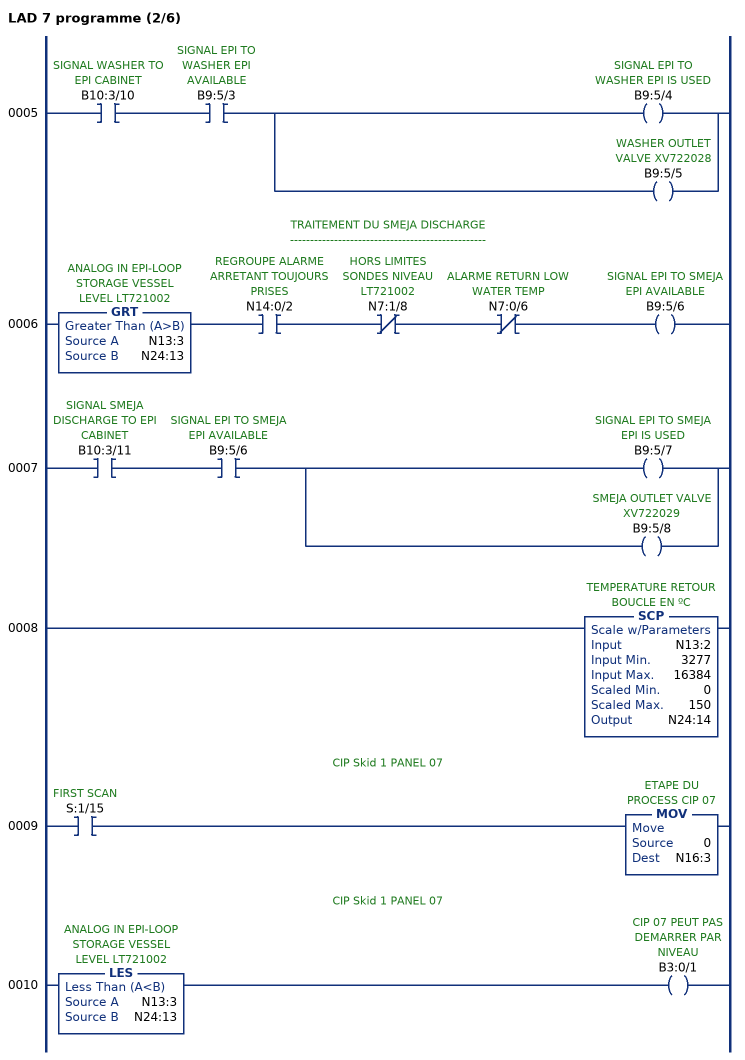
% Rung: 5 %
SOR XIC B10:3/10 XIC B9:5/3 BST OTE B9:5/4 NXB OTE B9:5/5 BND EOR
%   B10:3/10  "SIGNAL WASHER TO EPI CABINET" %
%   B9:5/3  "SIGNAL EPI TO WASHER EPI AVAILABLE" %
%   B9:5/4  "SIGNAL EPI TO WASHER EPI IS USED" %
%   B9:5/5  "WASHER OUTLET VALVE XV722028" %
% Rung: 6 %
% TRAITEMENT DU SMEJA DISCHARGE
% ------------------------------------------------- %
SOR GRT N13:3 N24:13 XIC N14:0/2 XIO N7:1/8 XIO N7:0/6 OTE B9:5/6 EOR
%   N13:3  "ANALOG IN EPI-LOOP STORAGE VESSEL LEVEL LT721002" %
%   N24:13  "LEVEL 5 LEVEL FROM LEVEL PROB AUTHORISE CIP+WASH.M" %
%   N14:0/2  "REGROUPE ALARME ARRETANT TOUJOURS PRISES" %
%   N7:1/8  "HORS LIMITES SONDES NIVEAU LT721002" %
%   N7:0/6  "ALARME RETURN LOW WATER TEMP" %
%   B9:5/6  "SIGNAL EPI TO SMEJA EPI AVAILABLE" %
% Rung: 7 %
SOR XIC B10:3/11 XIC B9:5/6 BST OTE B9:5/7 NXB OTE B9:5/8 BND EOR
%   B10:3/11  "SIGNAL SMEJA DISCHARGE TO EPI CABINET" %
%   B9:5/6  "SIGNAL EPI TO SMEJA EPI AVAILABLE" %
%   B9:5/7  "SIGNAL EPI TO SMEJA EPI IS USED" %
%   B9:5/8  "SMEJA OUTLET VALVE XV722029" %
% Rung: 8 %
SOR SCP N13:2 3277 16384 0 150 N24:14 EOR
%   N13:2  "ANALOG IN EPI-LOOP RETURN WATER TEMP TT722011" %
%   N24:14  "TEMPERATURE RETOUR BOUCLE EN ºC" %
% Rung: 9 %
% CIP Skid 1 PANEL 07 %
SOR XIC S:1/15 MOV 0 N16:3 EOR
%   S:1/15  "FIRST SCAN" %
%   N16:3  "ETAPE DU PROCESS CIP 07" %
% Rung: 10 %
% CIP Skid 1 PANEL 07 %
SOR LES N13:3 N24:13 OTE B3:0/1 EOR
%   N13:3  "ANALOG IN EPI-LOOP STORAGE VESSEL LEVEL LT721002" %
%   N24:13  "LEVEL 5 LEVEL FROM LEVEL PROB AUTHORISE CIP+WASH.M" %
%   B3:0/1  "CIP 07 PEUT PAS DEMARRER PAR NIVEAU" %

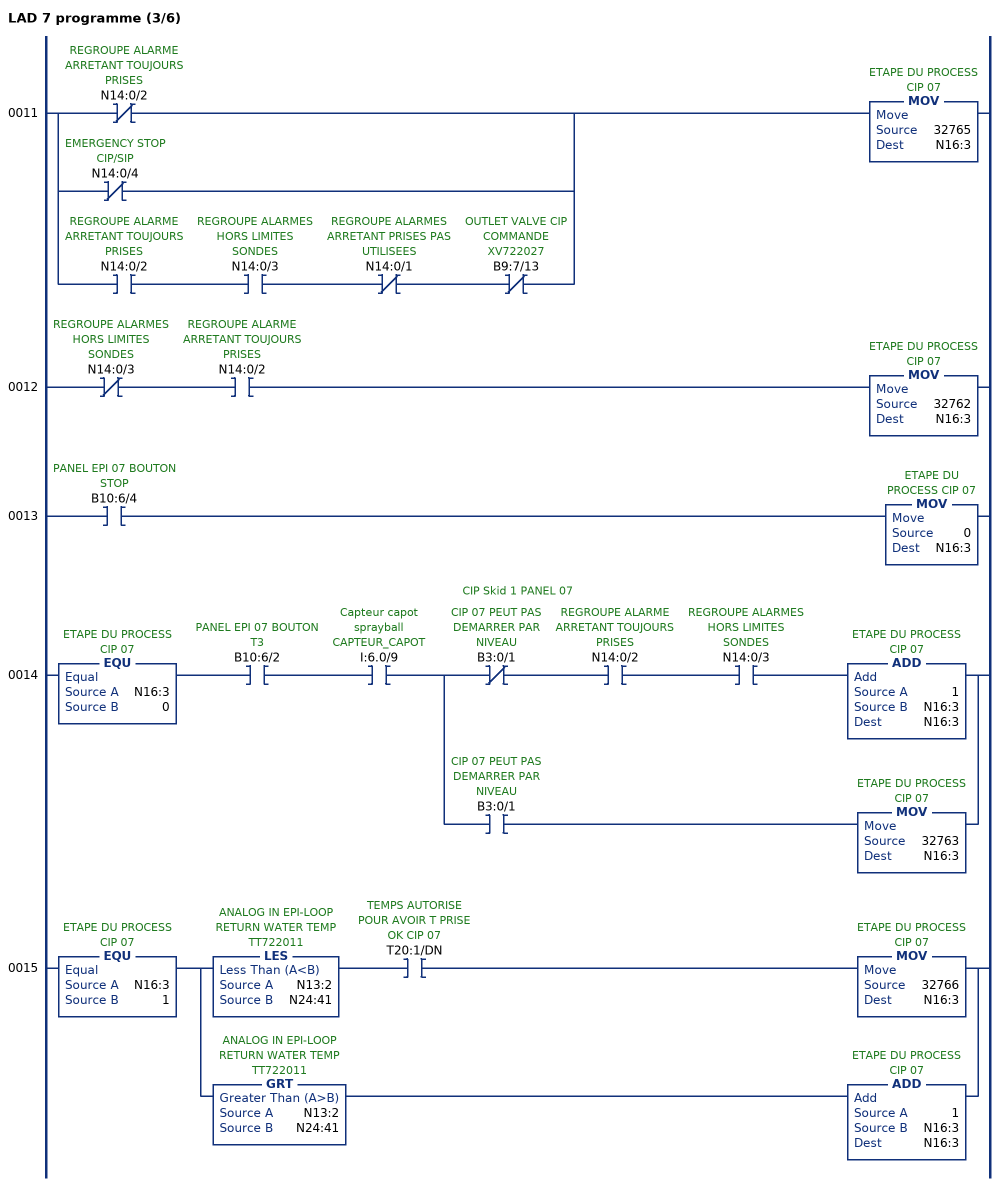
% Rung: 11 %
SOR BST BST XIO N14:0/2 NXB XIO N14:0/4 BND NXB XIC N14:0/2 XIC N14:0/3 XIO N14:0/1 XIO B9:7/13 BND MOV 32765 N16:3 EOR
%   N14:0/2  "REGROUPE ALARME ARRETANT TOUJOURS PRISES" %
%   N14:0/4  "EMERGENCY STOP CIP/SIP" %
%   N14:0/3  "REGROUPE ALARMES HORS LIMITES SONDES" %
%   N14:0/1  "REGROUPE ALARMES ARRETANT PRISES PAS UTILISEES" %
%   B9:7/13  "OUTLET VALVE CIP COMMANDE XV722027" %
%   N16:3  "ETAPE DU PROCESS CIP 07" %
% Rung: 12 %
SOR XIO N14:0/3 XIC N14:0/2 MOV 32762 N16:3 EOR
%   N14:0/3  "REGROUPE ALARMES HORS LIMITES SONDES" %
%   N14:0/2  "REGROUPE ALARME ARRETANT TOUJOURS PRISES" %
%   N16:3  "ETAPE DU PROCESS CIP 07" %
% Rung: 13 %
SOR XIC B10:6/4 MOV 0 N16:3 EOR
%   B10:6/4  "PANEL EPI 07 BOUTON STOP" %
%   N16:3  "ETAPE DU PROCESS CIP 07" %
% Rung: 14 %
% CIP Skid 1 PANEL 07 %
SOR EQU N16:3 0 XIC B10:6/2 XIC I:6.0/9 BST XIO B3:0/1 XIC N14:0/2 XIC N14:0/3 ADD 1 N16:3 N16:3 NXB XIC B3:0/1 MOV 32763 N16:3 BND EOR
%   N16:3  "ETAPE DU PROCESS CIP 07" %
%   B10:6/2  "PANEL EPI 07 BOUTON T3" %
%   I:6.0/9  CAPTEUR_CAPOT  "Capteur capot sprayball" %
%   B3:0/1  "CIP 07 PEUT PAS DEMARRER PAR NIVEAU" %
%   N14:0/2  "REGROUPE ALARME ARRETANT TOUJOURS PRISES" %
%   N14:0/3  "REGROUPE ALARMES HORS LIMITES SONDES" %
% Rung: 15 %
SOR EQU N16:3 1 BST LES N13:2 N24:41 XIC T20:1/DN MOV 32766 N16:3 NXB GRT N13:2 N24:41 ADD 1 N16:3 N16:3 BND EOR
%   N16:3  "ETAPE DU PROCESS CIP 07" %
%   N13:2  "ANALOG IN EPI-LOOP RETURN WATER TEMP TT722011" %
%   N24:41  "CONSIGNE T MINIMUM POUR DEMARRER CIP" %
%   T20:1/DN  "TEMPS AUTORISE POUR AVOIR T PRISE OK CIP 07" %

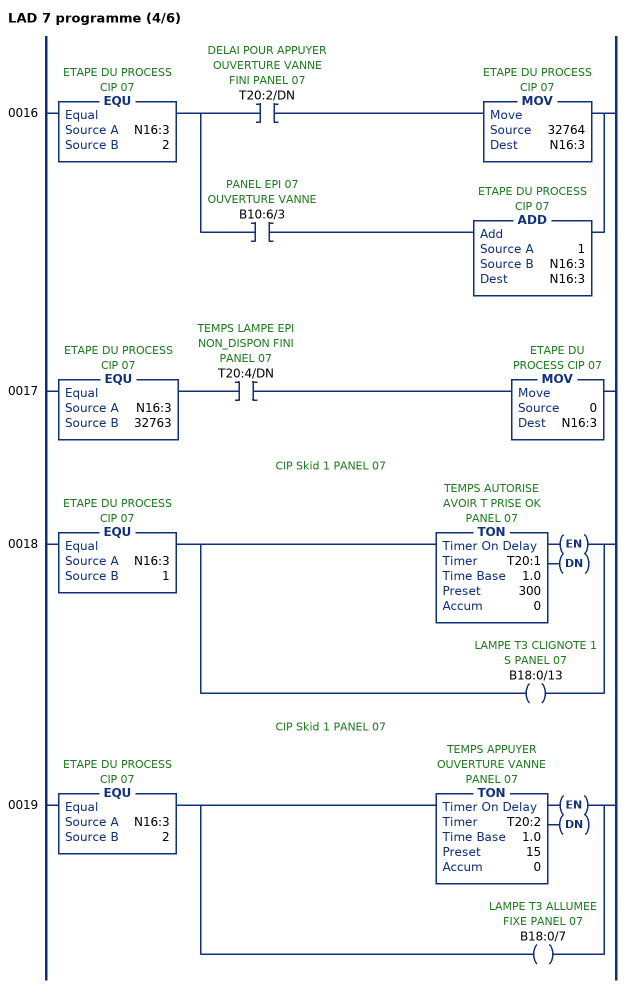
% Rung: 16 %
SOR EQU N16:3 2 BST XIC T20:2/DN MOV 32764 N16:3 NXB XIC B10:6/3 ADD 1 N16:3 N16:3 BND EOR
%   N16:3  "ETAPE DU PROCESS CIP 07" %
%   T20:2/DN  "DELAI POUR APPUYER OUVERTURE VANNE FINI PANEL 07" %
%   B10:6/3  "PANEL EPI 07 OUVERTURE VANNE" %
% Rung: 17 %
SOR EQU N16:3 32763 XIC T20:4/DN MOV 0 N16:3 EOR
%   N16:3  "ETAPE DU PROCESS CIP 07" %
%   T20:4/DN  "TEMPS LAMPE EPI NON_DISPON FINI PANEL 07" %
% Rung: 18 %
% CIP Skid 1 PANEL 07 %
SOR EQU N16:3 1 BST TON T20:1 1.0 300 0 NXB OTE B18:0/13 BND EOR
%   N16:3  "ETAPE DU PROCESS CIP 07" %
%   T20:1  "TEMPS AUTORISE AVOIR T PRISE OK PANEL 07" %
%   B18:0/13  "LAMPE T3 CLIGNOTE 1 S PANEL 07" %
% Rung: 19 %
% CIP Skid 1 PANEL 07 %
SOR EQU N16:3 2 BST TON T20:2 1.0 15 0 NXB OTE B18:0/7 BND EOR
%   N16:3  "ETAPE DU PROCESS CIP 07" %
%   T20:2  "TEMPS APPUYER OUVERTURE VANNE PANEL 07" %
%   B18:0/7  "LAMPE T3 ALLUMEE FIXE PANEL 07" %

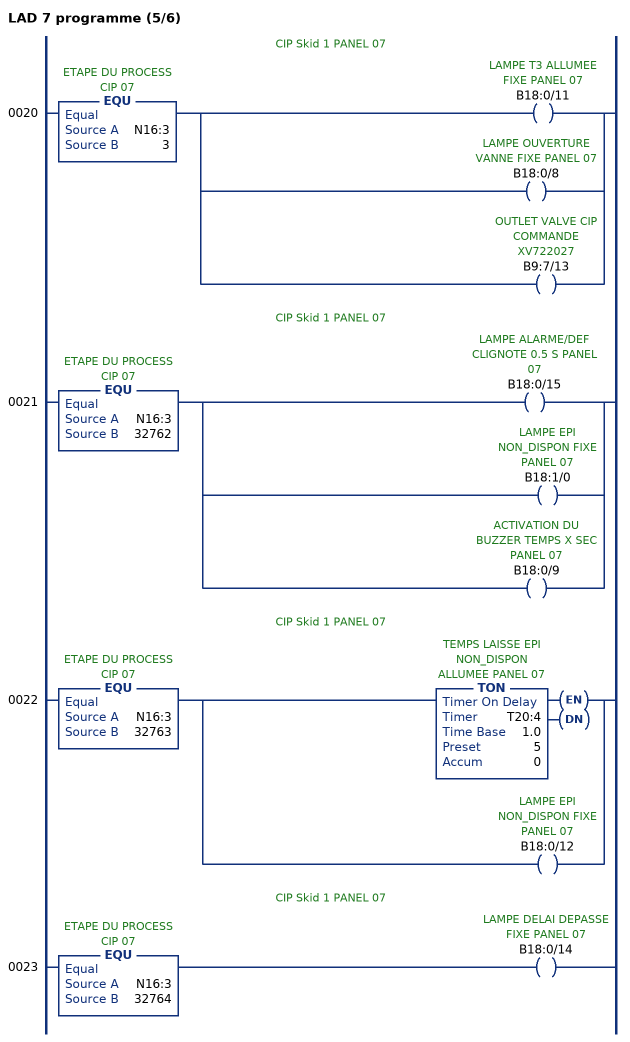
% Rung: 20 %
% CIP Skid 1 PANEL 07 %
SOR EQU N16:3 3 BST OTE B18:0/11 NXB OTE B18:0/8 NXB OTE B9:7/13 BND EOR
%   N16:3  "ETAPE DU PROCESS CIP 07" %
%   B18:0/11  "LAMPE T3 ALLUMEE FIXE PANEL 07" %
%   B18:0/8  "LAMPE OUVERTURE VANNE FIXE PANEL 07" %
%   B9:7/13  "OUTLET VALVE CIP COMMANDE XV722027" %
% Rung: 21 %
% CIP Skid 1 PANEL 07 %
SOR EQU N16:3 32762 BST OTE B18:0/15 NXB OTE B18:1/0 NXB OTE B18:0/9 BND EOR
%   N16:3  "ETAPE DU PROCESS CIP 07" %
%   B18:0/15  "LAMPE ALARME/DEF CLIGNOTE 0.5 S PANEL 07" %
%   B18:1/0  "LAMPE EPI NON_DISPON FIXE PANEL 07" %
%   B18:0/9  "ACTIVATION DU BUZZER TEMPS X SEC PANEL 07" %
% Rung: 22 %
% CIP Skid 1 PANEL 07 %
SOR EQU N16:3 32763 BST TON T20:4 1.0 5 0 NXB OTE B18:0/12 BND EOR
%   N16:3  "ETAPE DU PROCESS CIP 07" %
%   T20:4  "TEMPS LAISSE EPI NON_DISPON ALLUMEE PANEL 07" %
%   B18:0/12  "LAMPE EPI NON_DISPON FIXE PANEL 07" %
% Rung: 23 %
% CIP Skid 1 PANEL 07 %
SOR EQU N16:3 32764 OTE B18:0/14 EOR
%   N16:3  "ETAPE DU PROCESS CIP 07" %
%   B18:0/14  "LAMPE DELAI DEPASSE FIXE PANEL 07" %

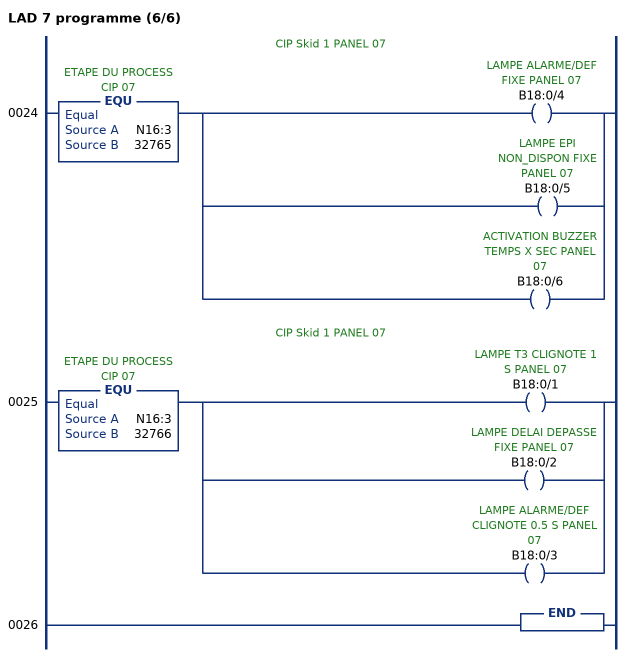
% Rung: 24 %
% CIP Skid 1 PANEL 07 %
SOR EQU N16:3 32765 BST OTE B18:0/4 NXB OTE B18:0/5 NXB OTE B18:0/6 BND EOR
%   N16:3  "ETAPE DU PROCESS CIP 07" %
%   B18:0/4  "LAMPE ALARME/DEF FIXE PANEL 07" %
%   B18:0/5  "LAMPE EPI NON_DISPON FIXE PANEL 07" %
%   B18:0/6  "ACTIVATION BUZZER TEMPS X SEC PANEL 07" %
% Rung: 25 %
% CIP Skid 1 PANEL 07 %
SOR EQU N16:3 32766 BST OTE B18:0/1 NXB OTE B18:0/2 NXB OTE B18:0/3 BND EOR
%   N16:3  "ETAPE DU PROCESS CIP 07" %
%   B18:0/1  "LAMPE T3 CLIGNOTE 1 S PANEL 07" %
%   B18:0/2  "LAMPE DELAI DEPASSE FIXE PANEL 07" %
%   B18:0/3  "LAMPE ALARME/DEF CLIGNOTE 0.5 S PANEL 07" %
% Rung: 26 %
SOR END EOR

LADDER 8 "pid"
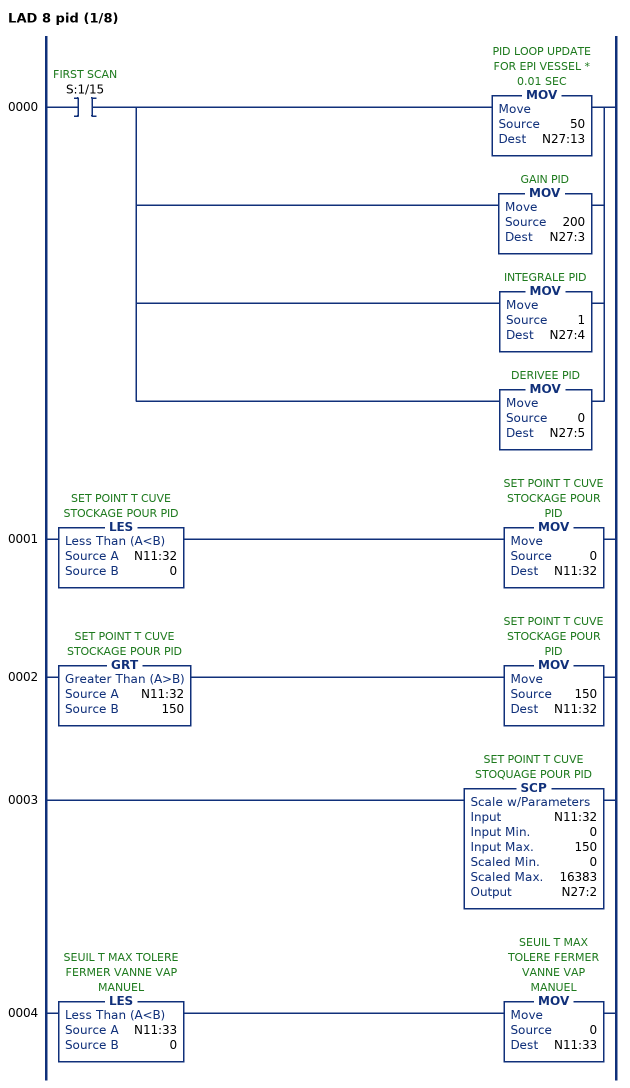
% Rung: 0 %
SOR XIC S:1/15 BST MOV 50 N27:13 NXB MOV 200 N27:3 NXB MOV 1 N27:4 NXB MOV 0 N27:5 BND EOR
%   S:1/15  "FIRST SCAN" %
%   N27:13  "PID LOOP UPDATE FOR EPI VESSEL * 0.01 SEC" %
%   N27:3  "GAIN PID" %
%   N27:4  "INTEGRALE PID" %
%   N27:5  "DERIVEE PID" %
% Rung: 1 %
SOR LES N11:32 0 MOV 0 N11:32 EOR
%   N11:32  "SET POINT T CUVE STOCKAGE POUR PID" %
% Rung: 2 %
SOR GRT N11:32 150 MOV 150 N11:32 EOR
%   N11:32  "SET POINT T CUVE STOCKAGE POUR PID" %
% Rung: 3 %
SOR SCP N11:32 0 150 0 16383 N27:2 EOR
%   N11:32  "SET POINT T CUVE STOCKAGE POUR PID" %
%   N27:2  "SET POINT T CUVE STOQUAGE POUR PID" %
% Rung: 4 %
SOR LES N11:33 0 MOV 0 N11:33 EOR
%   N11:33  "SEUIL T MAX TOLERE FERMER VANNE VAP MANUEL" %

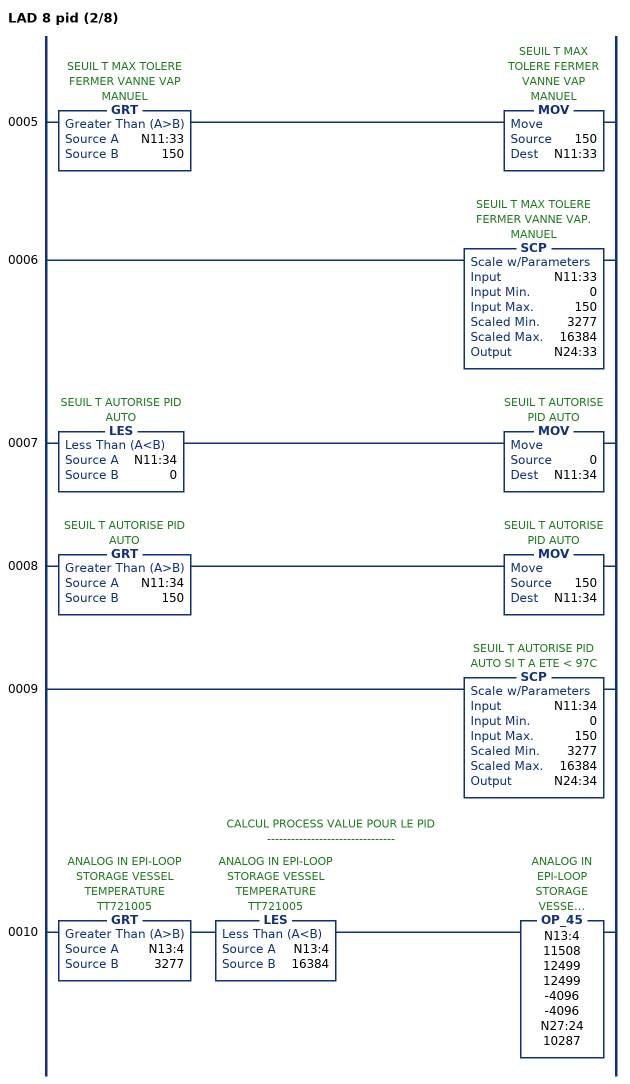
% Rung: 5 %
SOR GRT N11:33 150 MOV 150 N11:33 EOR
%   N11:33  "SEUIL T MAX TOLERE FERMER VANNE VAP MANUEL" %
% Rung: 6 %
SOR SCP N11:33 0 150 3277 16384 N24:33 EOR
%   N11:33  "SEUIL T MAX TOLERE FERMER VANNE VAP MANUEL" %
%   N24:33  "SEUIL T MAX TOLERE FERMER VANNE VAP. MANUEL" %
% Rung: 7 %
SOR LES N11:34 0 MOV 0 N11:34 EOR
%   N11:34  "SEUIL T AUTORISE PID AUTO" %
% Rung: 8 %
SOR GRT N11:34 150 MOV 150 N11:34 EOR
%   N11:34  "SEUIL T AUTORISE PID AUTO" %
% Rung: 9 %
SOR SCP N11:34 0 150 3277 16384 N24:34 EOR
%   N11:34  "SEUIL T AUTORISE PID AUTO" %
%   N24:34  "SEUIL T AUTORISE PID AUTO SI T A ETE < 97C" %
% Rung: 10 %
% CALCUL PROCESS VALUE POUR LE PID
% -------------------------------- %
SOR GRT N13:4 3277 LES N13:4 16384 OP_45 N13:4 11508 12499 12499 -4096 -4096 N27:24 10287 EOR
%   N13:4  "ANALOG IN EPI-LOOP STORAGE VESSEL TEMPERATURE TT721005" %
%   N27:24  "PROCESS VALUE T CUVE DU PID" %

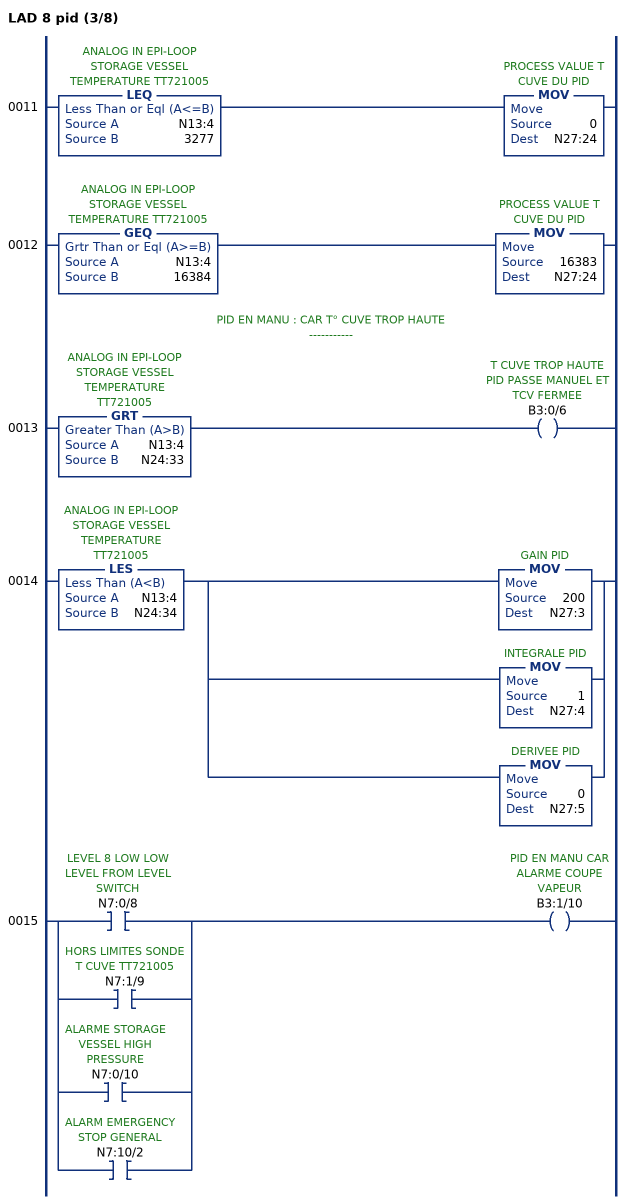
% Rung: 11 %
SOR LEQ N13:4 3277 MOV 0 N27:24 EOR
%   N13:4  "ANALOG IN EPI-LOOP STORAGE VESSEL TEMPERATURE TT721005" %
%   N27:24  "PROCESS VALUE T CUVE DU PID" %
% Rung: 12 %
SOR GEQ N13:4 16384 MOV 16383 N27:24 EOR
%   N13:4  "ANALOG IN EPI-LOOP STORAGE VESSEL TEMPERATURE TT721005" %
%   N27:24  "PROCESS VALUE T CUVE DU PID" %
% Rung: 13 %
% PID EN MANU : CAR T° CUVE TROP HAUTE
% ----------- %
SOR GRT N13:4 N24:33 OTE B3:0/6 EOR
%   N13:4  "ANALOG IN EPI-LOOP STORAGE VESSEL TEMPERATURE TT721005" %
%   N24:33  "SEUIL T MAX TOLERE FERMER VANNE VAP. MANUEL" %
%   B3:0/6  "T CUVE TROP HAUTE PID PASSE MANUEL ET TCV FERMEE" %
% Rung: 14 %
SOR LES N13:4 N24:34 BST MOV 200 N27:3 NXB MOV 1 N27:4 NXB MOV 0 N27:5 BND EOR
%   N13:4  "ANALOG IN EPI-LOOP STORAGE VESSEL TEMPERATURE TT721005" %
%   N24:34  "SEUIL T AUTORISE PID AUTO SI T A ETE < 97C" %
%   N27:3  "GAIN PID" %
%   N27:4  "INTEGRALE PID" %
%   N27:5  "DERIVEE PID" %
% Rung: 15 %
SOR BST XIC N7:0/8 NXB XIC N7:1/9 NXB XIC N7:0/10 NXB XIC N7:10/2 BND OTE B3:1/10 EOR
%   N7:0/8  "LEVEL 8 LOW LOW LEVEL FROM LEVEL SWITCH" %
%   N7:1/9  "HORS LIMITES SONDE T CUVE TT721005" %
%   N7:0/10  "ALARME STORAGE VESSEL HIGH PRESSURE" %
%   N7:10/2  "ALARM EMERGENCY STOP GENERAL" %
%   B3:1/10  "PID EN MANU CAR ALARME COUPE VAPEUR" %

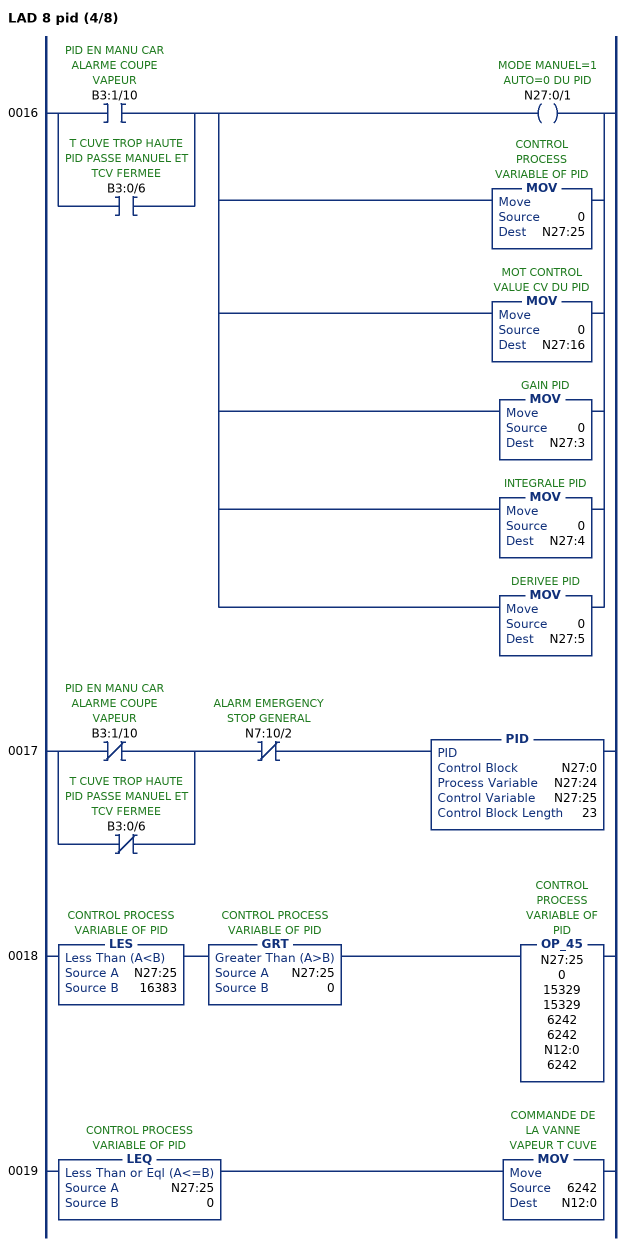
% Rung: 16 %
SOR BST XIC B3:1/10 NXB XIC B3:0/6 BND BST OTE N27:0/1 NXB MOV 0 N27:25 NXB BST MOV 0 N27:16 NXB MOV 0 N27:3 NXB MOV 0 N27:4 NXB MOV 0 N27:5 BND BND EOR
%   B3:1/10  "PID EN MANU CAR ALARME COUPE VAPEUR" %
%   B3:0/6  "T CUVE TROP HAUTE PID PASSE MANUEL ET TCV FERMEE" %
%   N27:0/1  "MODE MANUEL=1 AUTO=0 DU PID" %
%   N27:25  "CONTROL PROCESS VARIABLE OF PID" %
%   N27:16  "MOT CONTROL VALUE CV DU PID" %
%   N27:3  "GAIN PID" %
%   N27:4  "INTEGRALE PID" %
%   N27:5  "DERIVEE PID" %
% Rung: 17 %
SOR BST XIO B3:1/10 NXB XIO B3:0/6 BND XIO N7:10/2 PID N27:0 N27:24 N27:25 23 EOR
%   B3:1/10  "PID EN MANU CAR ALARME COUPE VAPEUR" %
%   B3:0/6  "T CUVE TROP HAUTE PID PASSE MANUEL ET TCV FERMEE" %
%   XIO B3:0/6  "T CUVE PAS TROP HAUTE ET TCV CUVE OUVERTE" %
%   N7:10/2  "ALARM EMERGENCY STOP GENERAL" %
%   N27:24  "PROCESS VALUE T CUVE DU PID" %
%   N27:25  "CONTROL PROCESS VARIABLE OF PID" %
% Rung: 18 %
SOR LES N27:25 16383 GRT N27:25 0 OP_45 N27:25 0 15329 15329 6242 6242 N12:0 6242 EOR
%   N27:25  "CONTROL PROCESS VARIABLE OF PID" %
%   N12:0  "COMMANDE DE LA VANNE VAPEUR T CUVE" %
% Rung: 19 %
SOR LEQ N27:25 0 MOV 6242 N12:0 EOR
%   N27:25  "CONTROL PROCESS VARIABLE OF PID" %
%   N12:0  "COMMANDE DE LA VANNE VAPEUR T CUVE" %

